// TIA Portal V17 export
// export: Created 2024-09-02T12:49:56.5704344Z, ExportSetting WithDefaults, DisplayName Totally Integrated Automation Portal, DisplayVersion V17, DisplayName TIA Portal Openness, DisplayVersion V17, DisplayName TIA Portal Version Control Interface, DisplayVersion V17, DisplayName STEP 7 Professional, DisplayVersion V17, DisplayName STEP 7 Safety, DisplayVersion V17, DisplayName WinCC Professional, DisplayVersion V17
FUNCTION_BLOCK "SysFB_HMI_SystemInit"   // FB259, LAD
TITLE = HMI system initialization / Initalisierung HMI-System
{ S7_Optimized_Access := 'TRUE' }
AUTHOR : OlegFuehrus
FAMILY : HMI
NAME : HMI
VERSION : 0.1
// stored: AutoNumber true, IsIECCheckEnabled false, IsRetainMemResEnabled false, MemoryReserve 100, SetENOAutomatically false, UDAEnableTagReadback false
   VAR_INPUT
      Start : Bool;
      DBNameS7G_Screen1_10 : WString[125];
      DBNameS7G_Screen11_20 : WString[125];
      DBNameS7G_Screen21_30 : WString[125];
      DBNameS7G_Screen31_40 : WString[125];
      DBNameS7G_Screen41_50 : WString[125];
      DBNameS7G_Screen51_58 : WString[125];
   END_VAR
   VAR_IN_OUT
      LTLL_Config : "LTLL_typeConfig";
      LTLL_Data : "LTLL_typeData";
      SYS_StepsHand : "TypeStepsHand";
      Finish : Bool;
   END_VAR
   VAR RETAIN
      s_Counter : Int;
      s_SNr : Int;
      s_Screen_Nr : Int;
      s_Screen_Counter : Int;
      s_INIT_ScreenConfig { S7_SetPoint := 'True'} : "LTLL_typeManualConfig";
      s_INIT_StepData { S7_SetPoint := 'True'} : "LTLL_typeManualData";
   END_VAR
   VAR_TEMP
      t_Counter : Int;
   END_VAR
BEGIN

REGION Network 1: INIT
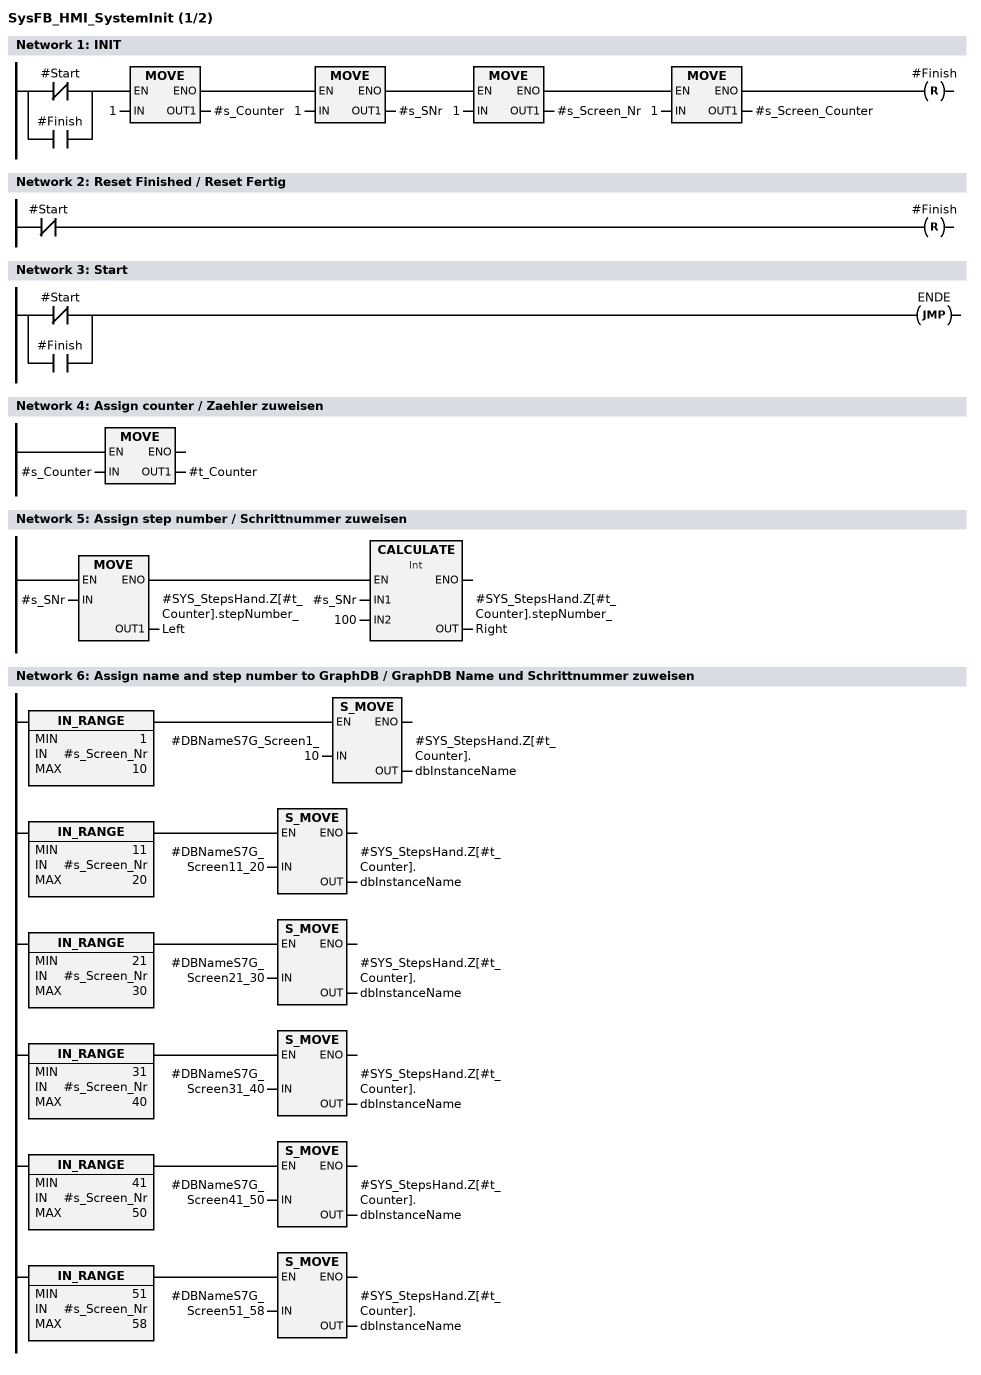
   RUNG wire#powerrail
      I_Contact( #Start )
      wire#w1
      Move(in := 1, out1 => #s_Counter)
      Move(in := 1, out1 => #s_SNr)
      Move(in := 1, out1 => #s_Screen_Nr)
      Move(in := 1, out1 => #s_Screen_Counter)
      R_Coil( #Finish )
   END_RUNG
   RUNG wire#powerrail
      Contact( #Finish )
   END_RUNG wire#w1
   // the same network as SCL:
   IF NOT #Start OR #Finish THEN
       #s_Counter := 1;
       #s_SNr := 1;
       #s_Screen_Nr := 1;
       #s_Screen_Counter := 1;
       #Finish := FALSE;
   END_IF;
END_REGION

REGION Network 2: Reset Finished / Reset Fertig
   RUNG wire#powerrail
      I_Contact( #Start )
      R_Coil( #Finish )
   END_RUNG
   // the same network as SCL:
   IF NOT #Start THEN #Finish := FALSE; END_IF;
END_REGION

REGION Network 3: Start
   RUNG wire#powerrail
      I_Contact( #Start )
      wire#w1
      JumpCoil( ENDE )
   END_RUNG
   RUNG wire#powerrail
      Contact( #Finish )
   END_RUNG wire#w1
   // the same network as SCL:
   IF NOT #Start OR #Finish THEN GOTO ENDE; END_IF;
END_REGION

REGION Network 4: Assign counter / Zaehler zuweisen
   RUNG wire#powerrail
      Move(in := #s_Counter, out1 => #t_Counter)
   END_RUNG
   // the same network as SCL:
   #t_Counter := #s_Counter;
END_REGION

REGION Network 5: Assign step number / Schrittnummer zuweisen
   RUNG wire#powerrail
      Move(in := #s_SNr, out1 => #SYS_StepsHand.Z[#t_Counter].stepNumber_Left)
      { S7_Templates := "SrcType := Int"; S7_Expression := "IN1 + IN2" } Calculate(in1 := #s_SNr, in2 := 100, out => #SYS_StepsHand.Z[#t_Counter].stepNumber_Right)
   END_RUNG
   // the same network as SCL:
   #SYS_StepsHand.Z[#t_Counter].stepNumber_Left := #s_SNr;
   #SYS_StepsHand.Z[#t_Counter].stepNumber_Right := #s_SNr + 100;
END_REGION

REGION Network 6: Assign name and step number to GraphDB / GraphDB Name und Schrittnummer zuweisen
   RUNG wire#powerrail
      { S7_Templates := "SrcType := Int" } InRange(min := 1, in := #s_Screen_Nr, max := 10)
      S_Move(in := #DBNameS7G_Screen1_10, out => #SYS_StepsHand.Z[#t_Counter].dbInstanceName)
   END_RUNG
   RUNG wire#powerrail
      { S7_Templates := "SrcType := Int" } InRange(min := 11, in := #s_Screen_Nr, max := 20)
      S_Move(in := #DBNameS7G_Screen11_20, out => #SYS_StepsHand.Z[#t_Counter].dbInstanceName)
   END_RUNG
   RUNG wire#powerrail
      { S7_Templates := "SrcType := Int" } InRange(min := 21, in := #s_Screen_Nr, max := 30)
      S_Move(in := #DBNameS7G_Screen21_30, out => #SYS_StepsHand.Z[#t_Counter].dbInstanceName)
   END_RUNG
   RUNG wire#powerrail
      { S7_Templates := "SrcType := Int" } InRange(min := 31, in := #s_Screen_Nr, max := 40)
      S_Move(in := #DBNameS7G_Screen31_40, out => #SYS_StepsHand.Z[#t_Counter].dbInstanceName)
   END_RUNG
   RUNG wire#powerrail
      { S7_Templates := "SrcType := Int" } InRange(min := 41, in := #s_Screen_Nr, max := 50)
      S_Move(in := #DBNameS7G_Screen41_50, out => #SYS_StepsHand.Z[#t_Counter].dbInstanceName)
   END_RUNG
   RUNG wire#powerrail
      { S7_Templates := "SrcType := Int" } InRange(min := 51, in := #s_Screen_Nr, max := 58)
      S_Move(in := #DBNameS7G_Screen51_58, out => #SYS_StepsHand.Z[#t_Counter].dbInstanceName)
   END_RUNG
   // the same network as SCL:
   IF (1 <= #s_Screen_Nr) AND (#s_Screen_Nr <= 10) THEN
       #SYS_StepsHand.Z[#t_Counter].dbInstanceName := #DBNameS7G_Screen1_10;
   END_IF;
   IF (11 <= #s_Screen_Nr) AND (#s_Screen_Nr <= 20) THEN
       #SYS_StepsHand.Z[#t_Counter].dbInstanceName := #DBNameS7G_Screen11_20;
   END_IF;
   IF (21 <= #s_Screen_Nr) AND (#s_Screen_Nr <= 30) THEN
       #SYS_StepsHand.Z[#t_Counter].dbInstanceName := #DBNameS7G_Screen21_30;
   END_IF;
   IF (31 <= #s_Screen_Nr) AND (#s_Screen_Nr <= 40) THEN
       #SYS_StepsHand.Z[#t_Counter].dbInstanceName := #DBNameS7G_Screen31_40;
   END_IF;
   IF (41 <= #s_Screen_Nr) AND (#s_Screen_Nr <= 50) THEN
       #SYS_StepsHand.Z[#t_Counter].dbInstanceName := #DBNameS7G_Screen41_50;
   END_IF;
   IF (51 <= #s_Screen_Nr) AND (#s_Screen_Nr <= 58) THEN
       #SYS_StepsHand.Z[#t_Counter].dbInstanceName := #DBNameS7G_Screen51_58;
   END_IF;
END_REGION

REGION Network 7: Initialization of HMI line images / Initalisierung HMI Zeilenbilder
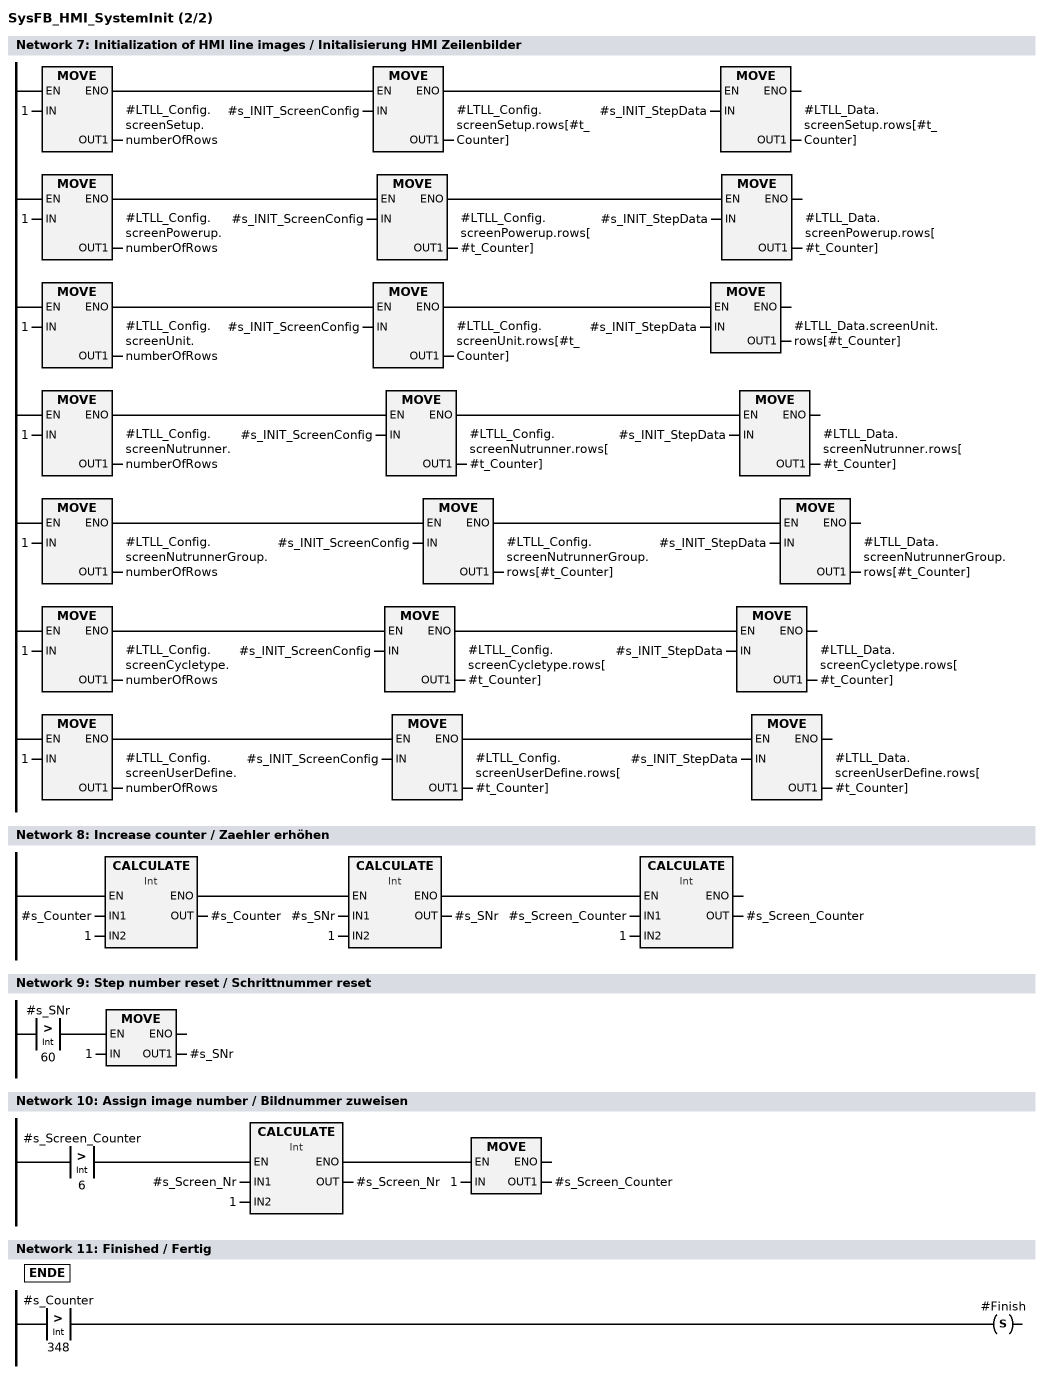
   RUNG wire#powerrail
      Move(in := 1, out1 => #LTLL_Config.screenSetup.numberOfRows)
      Move(in := #s_INIT_ScreenConfig, out1 => #LTLL_Config.screenSetup.rows[#t_Counter])
      Move(in := #s_INIT_StepData, out1 => #LTLL_Data.screenSetup.rows[#t_Counter])
   END_RUNG
   RUNG wire#powerrail
      Move(in := 1, out1 => #LTLL_Config.screenPowerup.numberOfRows)
      Move(in := #s_INIT_ScreenConfig, out1 => #LTLL_Config.screenPowerup.rows[#t_Counter])
      Move(in := #s_INIT_StepData, out1 => #LTLL_Data.screenPowerup.rows[#t_Counter])
   END_RUNG
   RUNG wire#powerrail
      Move(in := 1, out1 => #LTLL_Config.screenUnit.numberOfRows)
      Move(in := #s_INIT_ScreenConfig, out1 => #LTLL_Config.screenUnit.rows[#t_Counter])
      Move(in := #s_INIT_StepData, out1 => #LTLL_Data.screenUnit.rows[#t_Counter])
   END_RUNG
   RUNG wire#powerrail
      Move(in := 1, out1 => #LTLL_Config.screenNutrunner.numberOfRows)
      Move(in := #s_INIT_ScreenConfig, out1 => #LTLL_Config.screenNutrunner.rows[#t_Counter])
      Move(in := #s_INIT_StepData, out1 => #LTLL_Data.screenNutrunner.rows[#t_Counter])
   END_RUNG
   RUNG wire#powerrail
      Move(in := 1, out1 => #LTLL_Config.screenNutrunnerGroup.numberOfRows)
      Move(in := #s_INIT_ScreenConfig, out1 => #LTLL_Config.screenNutrunnerGroup.rows[#t_Counter])
      Move(in := #s_INIT_StepData, out1 => #LTLL_Data.screenNutrunnerGroup.rows[#t_Counter])
   END_RUNG
   RUNG wire#powerrail
      Move(in := 1, out1 => #LTLL_Config.screenCycletype.numberOfRows)
      Move(in := #s_INIT_ScreenConfig, out1 => #LTLL_Config.screenCycletype.rows[#t_Counter])
      Move(in := #s_INIT_StepData, out1 => #LTLL_Data.screenCycletype.rows[#t_Counter])
   END_RUNG
   RUNG wire#powerrail
      Move(in := 1, out1 => #LTLL_Config.screenUserDefine.numberOfRows)
      Move(in := #s_INIT_ScreenConfig, out1 => #LTLL_Config.screenUserDefine.rows[#t_Counter])
      Move(in := #s_INIT_StepData, out1 => #LTLL_Data.screenUserDefine.rows[#t_Counter])
   END_RUNG
   // the same network as SCL:
   #LTLL_Config.screenSetup.numberOfRows := 1;
   #LTLL_Config.screenSetup.rows[#t_Counter] := #s_INIT_ScreenConfig;
   #LTLL_Data.screenSetup.rows[#t_Counter] := #s_INIT_StepData;
   #LTLL_Config.screenPowerup.numberOfRows := 1;
   #LTLL_Config.screenPowerup.rows[#t_Counter] := #s_INIT_ScreenConfig;
   #LTLL_Data.screenPowerup.rows[#t_Counter] := #s_INIT_StepData;
   #LTLL_Config.screenUnit.numberOfRows := 1;
   #LTLL_Config.screenUnit.rows[#t_Counter] := #s_INIT_ScreenConfig;
   #LTLL_Data.screenUnit.rows[#t_Counter] := #s_INIT_StepData;
   #LTLL_Config.screenNutrunner.numberOfRows := 1;
   #LTLL_Config.screenNutrunner.rows[#t_Counter] := #s_INIT_ScreenConfig;
   #LTLL_Data.screenNutrunner.rows[#t_Counter] := #s_INIT_StepData;
   #LTLL_Config.screenNutrunnerGroup.numberOfRows := 1;
   #LTLL_Config.screenNutrunnerGroup.rows[#t_Counter] := #s_INIT_ScreenConfig;
   #LTLL_Data.screenNutrunnerGroup.rows[#t_Counter] := #s_INIT_StepData;
   #LTLL_Config.screenCycletype.numberOfRows := 1;
   #LTLL_Config.screenCycletype.rows[#t_Counter] := #s_INIT_ScreenConfig;
   #LTLL_Data.screenCycletype.rows[#t_Counter] := #s_INIT_StepData;
   #LTLL_Config.screenUserDefine.numberOfRows := 1;
   #LTLL_Config.screenUserDefine.rows[#t_Counter] := #s_INIT_ScreenConfig;
   #LTLL_Data.screenUserDefine.rows[#t_Counter] := #s_INIT_StepData;
END_REGION

REGION Network 8: Increase counter / Zaehler erhöhen
   RUNG wire#powerrail
      { S7_Templates := "SrcType := Int"; S7_Expression := "IN1 + IN2" } Calculate(in1 := #s_Counter, in2 := 1, out => #s_Counter)
      { S7_Templates := "SrcType := Int"; S7_Expression := "IN1 + IN2" } Calculate(in1 := #s_SNr, in2 := 1, out => #s_SNr)
      { S7_Templates := "SrcType := Int"; S7_Expression := "IN1 + IN2" } Calculate(in1 := #s_Screen_Counter, in2 := 1, out => #s_Screen_Counter)
   END_RUNG
   // the same network as SCL:
   #s_Counter := #s_Counter + 1;
   #s_SNr := #s_SNr + 1;
   #s_Screen_Counter := #s_Screen_Counter + 1;
END_REGION

REGION Network 9: Step number reset / Schrittnummer reset
   RUNG wire#powerrail
      { S7_Templates := "SrcType := Int" } GT_Contact(in1 := #s_SNr, in2 := 60)
      Move(in := 1, out1 => #s_SNr)
   END_RUNG
   // the same network as SCL:
   IF #s_SNr > 60 THEN #s_SNr := 1; END_IF;
END_REGION

REGION Network 10: Assign image number / Bildnummer zuweisen
   RUNG wire#powerrail
      { S7_Templates := "SrcType := Int" } GT_Contact(in1 := #s_Screen_Counter, in2 := 6)
      { S7_Templates := "SrcType := Int"; S7_Expression := "IN1 + IN2" } Calculate(in1 := #s_Screen_Nr, in2 := 1, out => #s_Screen_Nr)
      Move(in := 1, out1 => #s_Screen_Counter)
   END_RUNG
   // the same network as SCL:
   IF #s_Screen_Counter > 6 THEN
       #s_Screen_Nr := #s_Screen_Nr + 1;
       #s_Screen_Counter := 1;
   END_IF;
END_REGION

REGION Network 11: Finished / Fertig
   Label( ENDE )
   RUNG wire#powerrail
      { S7_Templates := "SrcType := Int" } GT_Contact(in1 := #s_Counter, in2 := 348)
      S_Coil( #Finish )
   END_RUNG
   // the same network as SCL:
   ENDE:
   IF #s_Counter > 348 THEN #Finish := TRUE; END_IF;
END_REGION

REGION Network 12: END / ENDE
END_REGION
END_FUNCTION_BLOCK
